TYPE typFBDOutput :
STRUCT
	xGate	: BOOL;
END_STRUCT
END_TYPE

(* stored: Version 1.1.0.1, ProductVersion 3.1.4024.6
   DUT typFBDOutput: Id {023ad5d8-88d1-4e7c-98e3-5c02a4206b6d} *)
